% RSLogix 500 project SARUUU_BAK010.RSS, saved by version 8.10.00.18 %
PROJECT "SARUUU"    % processor: MicroLogix 1200 %

PROGRAM FILES
  LAD 2   4 rungs

DATA FILES
  O0 OUTPUT  4 elements
  I1 INPUT  4 elements
  S2 STATUS  66 elements
  B3 BINARY  1 elements
  T4 TIMER  1 elements
  C5 COUNTER  1 elements
  R6 CONTROL  1 elements
  N7 INTEGER  1 elements

LADDER 2
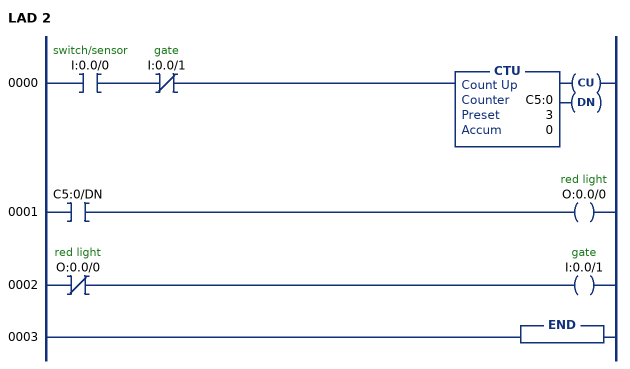
% Rung: 0 %
SOR XIC I:0.0/0 XIO I:0.0/1 CTU C5:0 3 0 EOR
%   I:0.0/0  "switch/sensor" %
%   I:0.0/1  "gate" %
% Rung: 1 %
SOR XIC C5:0/DN OTE O:0.0/0 EOR
%   O:0.0/0  "red light" %
% Rung: 2 %
SOR XIO O:0.0/0 OTE I:0.0/1 EOR
%   O:0.0/0  "red light" %
%   I:0.0/1  "gate" %
% Rung: 3 %
SOR END EOR

DATA TABLE (non-zero values as saved)
DATA C5
% .PRE .ACC %
% C5:0 % 3 0
